// TIA Portal V17 export
// export: Created 2026-04-13T11:12:44.5163412Z, ExportSetting WithDefaults, DisplayName Totally Integrated Automation Portal, DisplayVersion V17 Update 4, DisplayName TIA Portal Openness, DisplayVersion V17 Update 4, DisplayName TIA Portal Version Control Interface, DisplayVersion V17, DisplayName SINAMICS Startdrive Advanced, DisplayVersion V17, DisplayName SINAMICS Startdrive G130, G150, S120, S150, SINAMICS MV, S210, DisplayVersion V17, DisplayName SINAMICS Startdrive G110M, G120, G120C, G120D, G120P, G115D, DisplayVersion V17, DisplayName STEP 7 Professional, DisplayVersion V17 Update 4, DisplayName STEP 7 Safety, DisplayVersion V17, DisplayName WinCC Professional, DisplayVersion V17 Update 4
DATA_BLOCK "B3-全局连锁_DB"   // DB25
VERSION : 0.1
// stored: AutoNumber true, DBAccessibleFromOPCUA true, DBAccessibleFromWebserver true, InstanceOfName B3-全局连锁, InstanceOfType FB
"B3-全局连锁"
   // VAR
   //    T1S : TON_TIME;
   //    YC1 { S7_SetPoint := 'True'} : DInt;
   //    BJ报警上升辅助 : Bool;
   //    BJ报警下降辅助 : Bool;
   //    BJ报警上升沿 { S7_SetPoint := 'True'} : R_TRIG;
   //    BJ报警下降沿 { S7_SetPoint := 'True'} : F_TRIG;
   //    DH : Int;
   //    XT心跳上升沿延迟 : TON_TIME;
   //    XT心跳下降沿延迟 { S7_SetPoint := 'True'} : TON_TIME;
   // END_VAR
BEGIN
END_DATA_BLOCK
